FUNCTION_BLOCK CENTRALConCTL (* Basic Function Block Type *)
  (* Standard: 61499-2 *)
  (* Version 0.2, 2003-12-04, JHC, Rockwell Automation, Renamed for better indexing. *)
  (* Version 0.1, 2002-11-05, JHC, Rockwell Automation, Corrected missing ST element in Algorithm REQ. *)
  (* Version 0.0, 2000-05-30, JHC, Rockwell Automation *)
  (* Compiler header: package fb.rt.cs725; *)
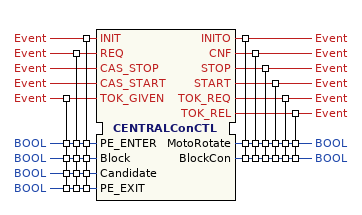
  EVENT_INPUT
    INIT WITH PE_ENTER, Block, Candidate, PE_EXIT; (* Initialization Request *)
    REQ WITH PE_ENTER, Block, Candidate, PE_EXIT; (* Normal Execution Request *)
    CAS_STOP;
    CAS_START;
    TOK_GIVEN WITH PE_ENTER, Block, PE_EXIT, Candidate;
  END_EVENT
  EVENT_OUTPUT
    INITO WITH MotoRotate, BlockCon; (* Initialization Confirm *)
    CNF WITH MotoRotate, BlockCon; (* Execution Confirmation *)
    STOP WITH MotoRotate, BlockCon;
    START WITH MotoRotate, BlockCon;
    TOK_REQ WITH MotoRotate, BlockCon;
    TOK_REL WITH MotoRotate, BlockCon;
  END_EVENT
  VAR_INPUT
    PE_ENTER : BOOL; (* Input event qualifier *)
    Block : BOOL;
    Candidate : BOOL;
    PE_EXIT : BOOL;
  END_VAR
  VAR_OUTPUT
    MotoRotate : BOOL; (* Output event qualifier *)
    BlockCon : BOOL;
  END_VAR
  VAR
    lastPE : BOOL := 1;
    lastBlock : BOOL := 0;
  END_VAR
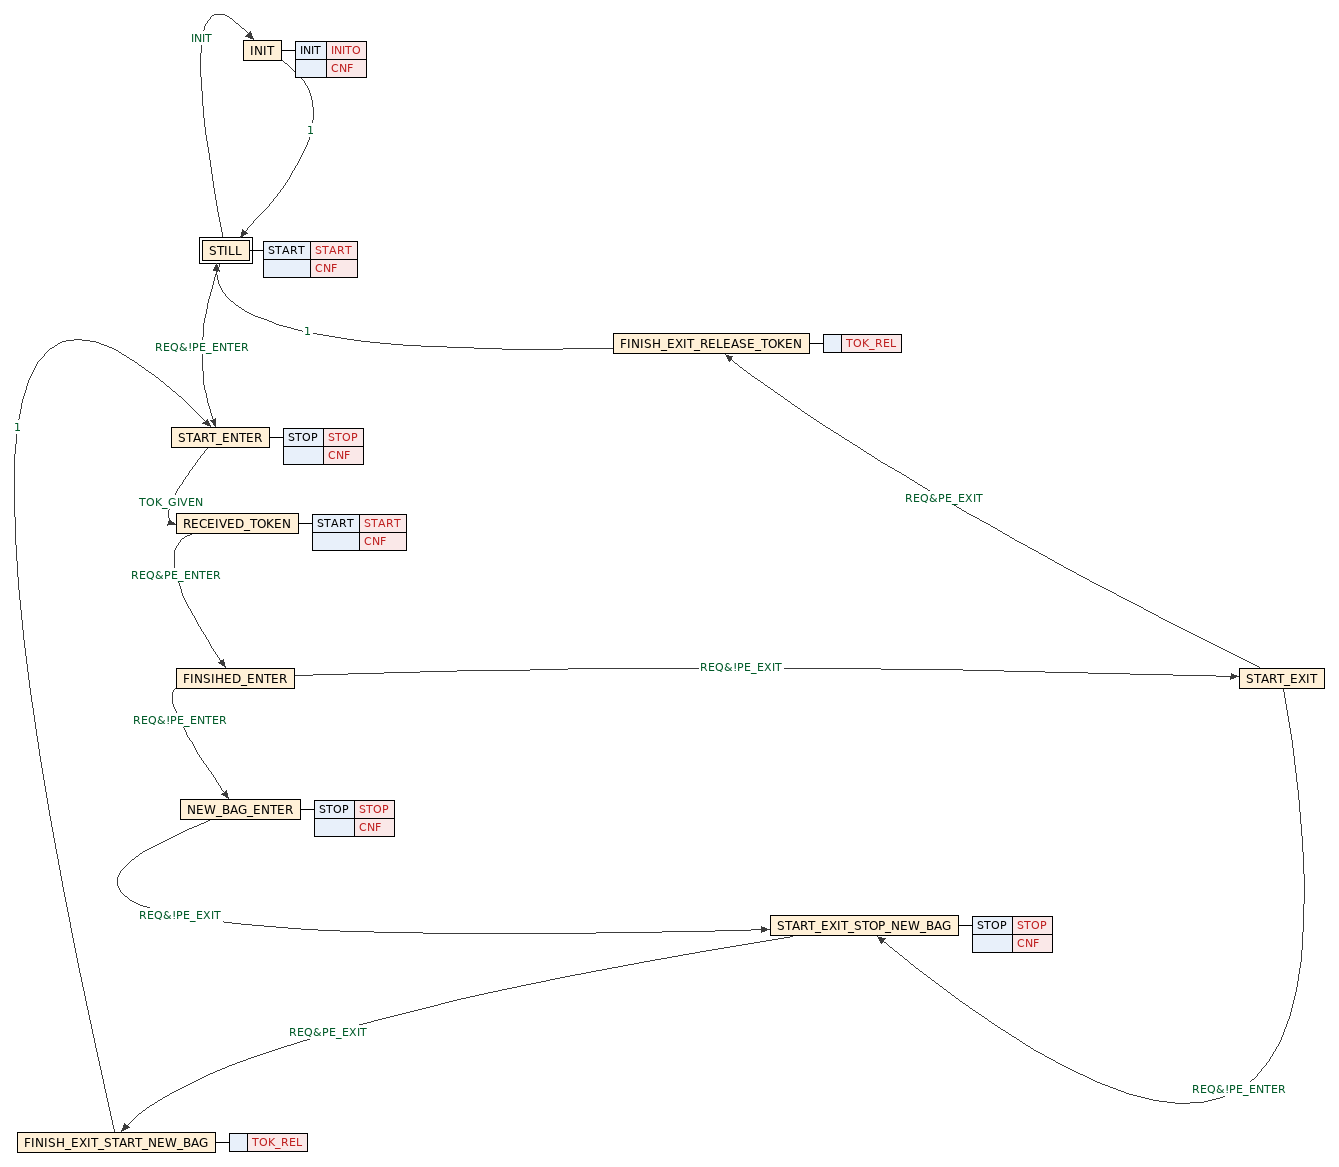
  EC_STATES
    STILL : START -> START, -> CNF; (* Initial State *)
    INIT : INIT -> INITO, -> CNF; (* Initialization *)
    START_ENTER : STOP -> STOP, -> CNF;
    RECEIVED_TOKEN : START -> START, -> CNF;
    NEW_BAG_ENTER : STOP -> STOP, -> CNF;
    FINSIHED_ENTER;
    START_EXIT;
    START_EXIT_STOP_NEW_BAG : STOP -> STOP, -> CNF;
    FINISH_EXIT_RELEASE_TOKEN : -> TOK_REL;
    FINISH_EXIT_START_NEW_BAG : -> TOK_REL;
  END_STATES
  EC_TRANSITIONS
    STILL TO INIT := INIT;
    INIT TO STILL := 1;
    START_ENTER TO RECEIVED_TOKEN := TOK_GIVEN;
    RECEIVED_TOKEN TO FINSIHED_ENTER := REQ&PE_ENTER;
    FINSIHED_ENTER TO NEW_BAG_ENTER := REQ&!PE_ENTER;
    NEW_BAG_ENTER TO START_EXIT_STOP_NEW_BAG := REQ&!PE_EXIT;
    FINSIHED_ENTER TO START_EXIT := REQ&!PE_EXIT;
    STILL TO START_ENTER := REQ&!PE_ENTER;
    FINISH_EXIT_RELEASE_TOKEN TO STILL := 1;
    START_EXIT TO FINISH_EXIT_RELEASE_TOKEN := REQ&PE_EXIT;
    FINISH_EXIT_START_NEW_BAG TO START_ENTER := 1;
    START_EXIT_STOP_NEW_BAG TO FINISH_EXIT_START_NEW_BAG := REQ&PE_EXIT;
    START_EXIT TO START_EXIT_STOP_NEW_BAG := REQ&!PE_ENTER;
  END_TRANSITIONS
  ALGORITHM INIT IN ST: (* Initialization algorithm *)
MotoRotate := TRUE;
Block := FALSE;

System.out.println(this + " " + MotoRotate);
System.out.println(MotoRotate);
  END_ALGORITHM
  ALGORITHM REQ IN ST: (* Normally executed algorithm *)
System.out.println(this +  " -> Candidate" + Candidate);
IF Candidate THEN
IF lastPE !:= PE_ENTER THEN
IF NOT PE_ENTER THEN
BlockCon:= TRUE;
System.out.println("BlockCon = true");
ELSE
BlockCon:=FALSE;
System.out.println("BlockCon = false");
END_IF
lastPE := PE_ENTER;
END_IF
IF lastBlock !:= Block THEN
IF Block THEN
STOP.serviceEvent(this);
MotoRotate := FALSE;
System.out.println("Cas Stop");
ELSE
START.serviceEvent(this);
MotoRotate := TRUE;
System.out.println("Cas Start");
END_IF
lastBlock := Block;
END_IF
END_IF
  END_ALGORITHM
  ALGORITHM START IN ST:
MotoRotate:=TRUE;
System.out.println(this + " Start " + MotoRotate);

System.out.println("Start " + MotoRotate);
  END_ALGORITHM
  ALGORITHM STOP IN ST:
MotoRotate := FALSE;
System.out.println(this + " Stop " + MotoRotate);

System.out.println("Stop " + MotoRotate);
  END_ALGORITHM
END_FUNCTION_BLOCK
